//==================================================================================================
//							Beckhoff Automation Poland
//									11.04.2018
//	This object shall provide the text id of the last DiagMessage of type error, which occurred in this axis.
//  v1.0	|| TC v 3.1.4022.16		|| - pierwsza wersja
//==================================================================================================
FUNCTION_BLOCK FB_ReadChannelErrorCodeAX8000
VAR_INPUT
	bExecute 						: BOOL;
	stDriveRef						: ST_DriveRef;						// 
END_VAR
VAR_OUTPUT
	bBusy							: BOOL;
	bError							: BOOL; 							// General error: parameter or CoE read.
	iAdsErrId						: UINT;								// Forwarded output FB_CoERead_ByDriveRef
	iCANopenErrId					: UINT;								// Forwarded output FB_CoERead_ByDriveRef
	uiChannelErrorCode				: UINT;								// 603F Error code	0x603F (Ch A)/ 0x683F (Ch B) 	UINT16
	{attribute 'displaymode':='hex'}
	uiChannelErrorCodeHex			: UINT;								// 603F Error code	0x603F (Ch A)/ 0x683F (Ch B) 	UINT16
END_VAR
VAR
	fbCoERead						: FB_CoERead_ByDriveRef;			// FB for read CoE parameters
END_VAR

fbCoERead(	stDriveRef					:= stDriveRef,
			nIndex						:= 16#603F + (stDriveRef.nDriveNo * 16#800),
			nSubIndex					:= 0,
			pDstBuf						:= ADR(uiChannelErrorCode),
			cbBufLen					:= SIZEOF(uiChannelErrorCode),
			bExecute					:= bExecute,
			bBusy						=> bBusy,
			bError						=> bError,
			iAdsErrId					=> iAdsErrId,
			iCANopenErrId				=> iCANopenErrId);

uiChannelErrorCodeHex					:= uiChannelErrorCode;

END_FUNCTION_BLOCK

(* stored: Version 1.1.0.1, ProductVersion 3.1.4022.12
   POU FB_ReadChannelErrorCodeAX8000: Id {449892ff-9e2a-4827-a4c7-2bb2ca0bb142}, SpecialFunc None *)
